VAR_GLOBAL
END_VAR

(* stored: Version 1.1.0.1, ProductVersion 3.1.0.12
   GVL Variable_Configuration: Id {49fe29e9-282a-4c4b-b3af-8056c7c12783} *)
